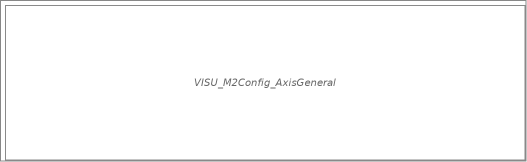
VISUALIZATION VISU_M2Config_PotentiometerAxis  // 527x162
VAR_IN_OUT
    editable : M2PotentiometerAxisConfig;
	active : M2PotentiometerAxisConfig;
END_VAR
    Frame (5,5 520x155)
        shows VISU_M2Config_AxisGeneral(editable := editable.general, active := active.general)
END_VISUALIZATION

(* stored: Version 1.1.0.1, ProductVersion 3.1.4019.2
   Visu VISU_M2Config_PotentiometerAxis: Id {b4b4f712-ba59-400c-9a11-69d239f2f8e8} *)
